// TIA Portal V20 export
DATA_BLOCK "Instace_FB_Search_Water_Foutain_DB"   // DB109
// stored: AutoNumber false, InstanceOfName FB_Search_Water_Foutain, InstanceOfType FB
"FB_Search_Water_Foutain"
   // VAR_INPUT
   //    Trigger_Read_Serial_Number_Exit_Functional_Test : Bool;
   //    Serial_Number : String[17];
   //    Functional_Tests_Panels : Array[0..31] of "Functional_Test";
   // END_VAR
   // VAR_OUTPUT
   //    Found_Functional_Test : Bool;
   //    Water_Foutain_Fail_Functional_Test : Bool;
   //    DataLog_Write : Bool;
   //    i : SInt;
   //    Search_Functional_Test : "Functional_Test";
   //    Reset_PLC_Functional_Test : Array[0..31] of Bool;
   // END_VAR
   // VAR
   //    Timer_Delay_Write_DataLog { S7_SetPoint := 'True'} : TON_TIME;
   // END_VAR
BEGIN
END_DATA_BLOCK
